# EPICS autosave request: softGlueApp/Db/clockConfig_settings.req
#$(P)$(H)clock1desiredFreq
$(P)$(H)clock2desiredFreq
$(P)$(H)clock3desiredFreq
$(P)$(H)clock4desiredFreq
$(P)$(H)clock5desiredFreq
$(P)$(H)clock6desiredFreq
